Staubli VAL3: getListItem.pgx

public program getListItem(string& x_sItem[], num x_nIndex)
begin
  //
  // define the item to show in the edit page Traj
  // customize an array and copy to x_sItem...
  //
  // see other traj as example

end
